{attribute 'no_check'}
//Publisher/Subscriber IOs
FUNCTION_BLOCK EAP_PUB_SUB_IO 
VAR_OUTPUT CONSTANT
END_VAR
VAR_INPUT
	{attribute 'displaymode':='hex'}
	FrameCtrl									AT %Q*:	UINT;
END_VAR		
VAR_OUTPUT	
	{attribute 'displaymode':='hex'}
	FrameState									AT %I*:	UINT;
	
	NotSentFrameSkipped								: Bool;
	ErrorFrameOversized								: Bool;
	SubscriberMissing								: Bool;
END_VAR
VAR
END_VAR

	(* IOs 									*)
	(****************************************)

(* Read status *****************************************)
	NotSentFrameSkipped						:= FrameState.0;
	ErrorFrameOversized						:= FrameState.1;
	SubscriberMissing						:= FrameState.2;

(*******************************************************)

PROPERTY PUBLIC disableSending : BOOL
GET
disableSending		:= FrameCtrl.1;
END_GET
SET
FrameCtrl.1				:= disableSending;
END_SET
END_PROPERTY

PROPERTY PUBLIC removeDestMacFromARPCache : BOOL
GET
RemoveDestMacFromARPCache		:= FrameCtrl.1;
END_GET
SET
FrameCtrl.1				:= RemoveDestMacFromARPCache;
END_SET
END_PROPERTY

END_FUNCTION_BLOCK

(* stored: Version 1.1.0.1, ProductVersion 3.1.4024.12
   POU EAP_PUB_SUB_IO: Id {7453658e-208e-4bcc-9617-517d78295e6f}, SpecialFunc None
   Property disableSending: Id {abf4973d-dcc7-4e61-8527-414d6fa86bb1}
   Get Get: Id {4ffa6b3a-8ffb-4f35-bf1d-306bd930374e}
   Set Set: Id {07f9fc1b-f32d-42d8-800b-c0bd2a640d5c}
   Property removeDestMacFromARPCache: Id {cfa48344-16e2-440f-b25b-79d2c3f4a35c}
   Get Get: Id {767ada1f-dd21-4c38-9612-70f352a1ced6}
   Set Set: Id {565655ba-1d15-43aa-93f6-0658bc3713af} *)
